% RSLogix 500 project Q11.RSS, saved by version 8.30.00.16 %
PROJECT "Q11"    % processor: Bul.1763 MicroLogix 1100 Series B %

PROGRAM FILES
  LAD 2   4 rungs

DATA FILES
  O0 OUTPUT  4 elements
  I1 INPUT  6 elements
  S2 STATUS  66 elements
  B3 BINARY  1 elements
  T4 TIMER  1 elements
  C5 COUNTER  1 elements
  R6 CONTROL  1 elements
  N7 INTEGER  1 elements
  F8 FLOAT  1 elements

LADDER 2
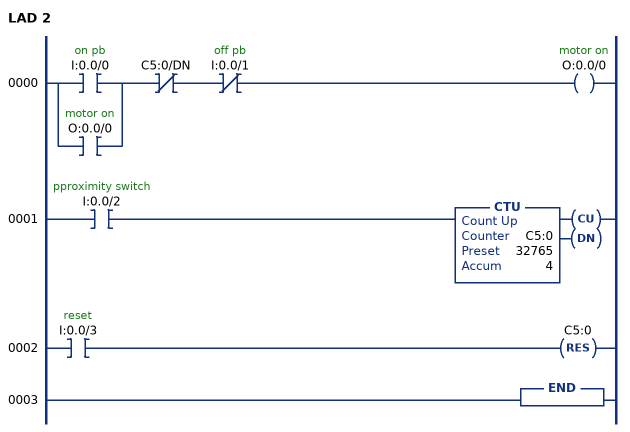
% Rung: 0 %
SOR BST XIC I:0.0/0 NXB XIC O:0.0/0 BND XIO C5:0/DN XIO I:0.0/1 OTE O:0.0/0 EOR
%   I:0.0/0  "on pb" %
%   O:0.0/0  "motor on" %
%   I:0.0/1  "off pb" %
% Rung: 1 %
SOR XIC I:0.0/2 CTU C5:0 32765 4 EOR
%   I:0.0/2  "pproximity switch" %
% Rung: 2 %
SOR XIC I:0.0/3 RES C5:0 EOR
%   I:0.0/3  "reset" %
% Rung: 3 %
SOR END EOR

DATA TABLE (non-zero values as saved)
DATA C5
% .PRE .ACC %
% C5:0 % 32765 4
